TEXTLIST ErrorList1
  1 = 'Az NTC vágó foglalt!'
  3 = 'A hajlítók nem állnak készen, vagy nem érkezett meg a szán az előhajlításhoz.'
  4 = 'Nem végzett idöben az elöhajlító.'
  6 = 'Nem érkezett meg a szán a véghajlításhoz.'
  7 = 'Nem állnak készen a hajlítók.'
  8 = 'Nem végzett a véghajlító.'
  10 = 'Nem érkezett meg a szán az első hegesztéshez.'
  12 = 'Nem érkezett meg az 1. hegesztésnél a fej.'
  13 = 'Nem lett kész az 1. hegesztési folyamat.'
  15 = 'Nem húzódott vissza az 1. hegesztésnél a fej.'
  16 = 'Nem érkezett meg a szán a 3. hegesztéshez.'
  18 = 'Nem érkezett meg a 3. hegesztésnél a fej.'
  19 = 'Nem lett kész a 3. hegesztési folyamat.'
  21 = 'Nem húzódott vissza a 3. hegesztésnél a fej.'
  22 = 'Nem érkezett meg a szán a 2. hegesztéshez.'
  24 = 'Nem érkezett meg a 2. hegesztésnél a fej.'
  25 = 'Nem lett kész a 2. hegesztési folyamat.'
  27 = 'Nem húzódott vissza a 2. hegesztésnél a fej.'
  28 = 'Nem érkezett meg a szán a 4. hegesztéshez.'
  29 = 'Nem fejeződött be az NTC vágás.'
  32 = 'Nem áll rendelkezésre a robot vagy nincs levágva az NTC.'
  33 = 'A megfogó nem engedte el a levágott NTC-t.'
  34 = 'A robot még nem vitte oda az NTC-t a hegesztéshez, vagy foglalt a hegesztő.'
  36 = 'Nem érkezett meg a 4. hegesztésnél a fej.'
  37 = 'Nem lett kész a 4. hegesztési folyamat.'
  39 = 'Nem húzódott vissza a 4. hegesztésnél a fej.'
  41 = 'A robot még nem jött el a hegesztés helyétől.'
  42 = 'Nem érkezett meg a szán az 5. hegesztéshez.'
  44 = 'Nem érkezett meg az 5. hegesztésnél a fej.'
  45 = 'Nem lett kész az 5. hegesztési folyamat.'
  47 = 'Nem húzódott vissza az 5. hegesztésnél a fej.'
  110 = 'Nem fejeződött be az NTC vágás.'
  112 = 'Az NTC vágó foglalt.'
  113 = 'Nem fejeződött be az NTC vágás.'
   = ''
END_TEXTLIST

(* stored: Version 1.1.0.1, ProductVersion 3.1.4020.3
   TextList ErrorList1: Id {34b58379-d64a-4154-b41b-44a9c00c482c} *)
